(* Base of Hardware Observations. Ideally, this is the base of every Hardware Control FB. *)
FUNCTION_BLOCK ABSTRACT HardwareObservationBase
VAR
END_VAR

METHOD ABSTRACT ResetDefinition : BOOL
VAR_INPUT
END_VAR
END_METHOD

(* Update an instance of ProcessState with the part of the process that can be observed by this Hardware Interface. *)
METHOD ABSTRACT UpdateProcessObservation : BOOL
VAR_IN_OUT
	io_processState: ProcessState;
END_VAR
END_METHOD

END_FUNCTION_BLOCK

(* stored: Version 1.1.0.1, ProductVersion 3.1.4024.12
   POU HardwareObservationBase: Id {6736ee86-4fb8-40de-8ddf-be9c37d4b4db}, SpecialFunc None
   Method ResetDefinition: Id {d4ba8c7a-263a-47c1-ba2b-ae132a94e35e}
   Method UpdateProcessObservation: Id {5c0aea51-22cd-4b0a-92cc-552ce94676ac} *)
